(* CODESYS project Visualization.vis.xml

Project tree, tasks and I/O mapping:
  visualisation Visualization
*)

// /Visualization
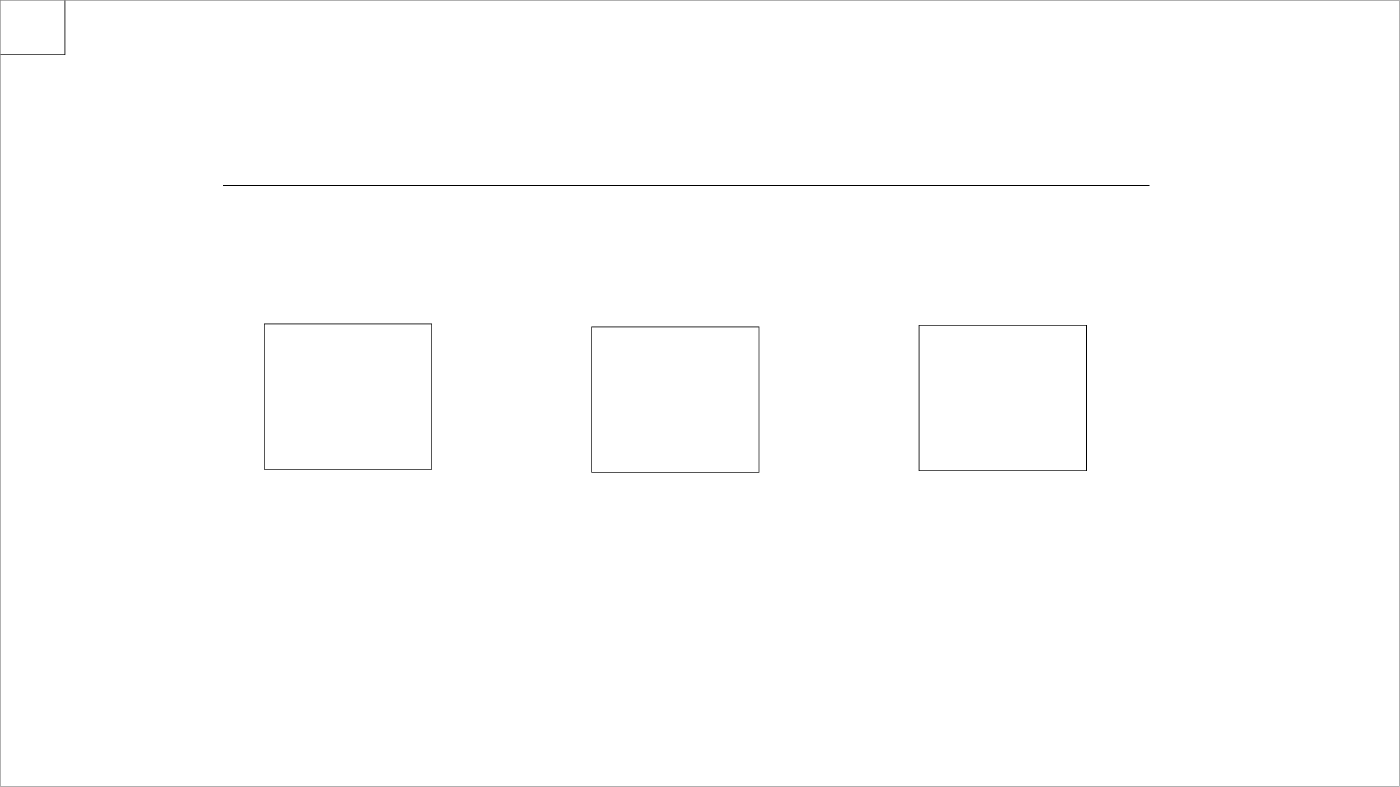
VISUALIZATION Visualization  // 1920x1080
    Line (306,254) (1576,254)
    Rectangle (362,444 230x200)
    Rectangle (811,448 230x200)
    Rectangle (1260,446 230x200)
    Rectangle (0,0 89x75)
        p3560616238: GVL_HMI.HMI.ActualX
        p2738717112: GVL_HMI.HMI.ActualZ
END_VISUALIZATION
